FUNCTION_BLOCK FB_FastFault
VAR_INPUT
END_VAR
VAR_OUTPUT
END_VAR
VAR
END_VAR

END_FUNCTION_BLOCK

(* stored: Version 1.1.0.1, ProductVersion 3.1.4022.12
   POU FB_FastFault: Id {a7225e03-a5d8-094a-35f2-8e6e41471d21}, SpecialFunc None *)
